LIN {X 0,Y 87.51,Z 409.05,A -85,B 0,C 180,E1 -30606.359,E2 -30606.359} C_VEL
LIN {X 0,Y 79.775,Z 420.472,A -85,B 0,C 180,E1 -30607.649,E2 -30607.649} C_VEL
LIN {X 0,Y 71.234,Z 430.536,A -85,B 0,C 180,E1 -30609.388,E2 -30609.388} C_VEL
LIN {X 0,Y 62.803,Z 438.788,A -85,B 0,C 180,E1 -30611.717,E2 -30611.717} C_VEL
LIN {X 0,Y 52.393,Z 447.262,A -85,B 0,C 180,E1 -30615.825,E2 -30615.825} C_VEL
LIN {X 0,Y 44.908,Z 452.36,A -85,B 0,C 180,E1 -30620.118,E2 -30620.118} C_VEL
LIN {X 0,Y 35.789,Z 457.715,A -85,B 0,C 180,E1 -30627.912,E2 -30627.912} C_VEL
LIN {X 0,Y 27.714,Z 461.88,A -85,B 0,C 180,E1 -30640.469,E2 -30640.469} C_VEL
LIN {X 0,Y 23.498,Z 464.077,A -85,B 0,C 180,E1 -30653.261,E2 -30653.261} C_VEL
LIN {X 0,Y 20.749,Z 465.788,A -85,B 0,C 180,E1 -30670.202,E2 -30670.202} C_VEL
LIN {X 0,Y 20.019,Z 467.089,A -85,B 0,C 180,E1 -30690.001,E2 -30690.001} C_VEL
LIN {X 0,Y 20.814,Z 467.966,A -85,B 0,C 180,E1 -30709.735,E2 -30709.735} C_VEL
LIN {X 0,Y 23.568,Z 468.43,A -85,B 0,C 180,E1 -30726.614,E2 -30726.614} C_VEL
LIN {X 0,Y 33.054,Z 468.146,A -85,B 0,C 180,E1 -30748.265,E2 -30748.265} C_VEL
LIN {X 0,Y 45.111,Z 466.339,A -85,B 0,C 180,E1 -30759.192,E2 -30759.192} C_VEL
LIN {X 0,Y 51.526,Z 464.795,A -85,B 0,C 180,E1 -30762.705,E2 -30762.705} C_VEL
LIN {X 0,Y 63.326,Z 460.995,A -85,B 0,C 180,E1 -30767.176,E2 -30767.176} C_VEL
LIN {X 0,Y 74.89,Z 455.966,A -85,B 0,C 180,E1 -30770.187,E2 -30770.187} C_VEL
LIN {X 0,Y 86.865,Z 449.183,A -85,B 0,C 180,E1 -30772.354,E2 -30772.354} C_VEL
LIN {X 0,Y 97.233,Z 441.823,A -85,B 0,C 180,E1 -30773.643,E2 -30773.643} C_VEL
LIN {X 0,Y 107.631,Z 432.702,A -85,B 0,C 180,E1 -30774.735,E2 -30774.735} C_VEL
LIN {X 0,Y 116.334,Z 423.229,A -85,B 0,C 180,E1 -30775.417,E2 -30775.417} C_VEL
LIN {X 0,Y 124.178,Z 412.736,A -85,B 0,C 180,E1 -30775.957,E2 -30775.957} C_VEL
LIN {X 0,Y 131.301,Z 400.788,A -85,B 0,C 180,E1 -30776.367,E2 -30776.367} C_VEL
LIN {X 0,Y 134.706,Z 393.665,A -85,B 0,C 180,E1 -30776.626,E2 -30776.626} C_VEL
LIN {X 0,Y 135.001,Z 392.963,A -85,B 0,C 180,E1 -30777.016,E2 -30777.016} C_VEL
LIN {X 0,Y 134.921,Z 393.119,A -85,B 0,C 180,E1 -30777.835,E2 -30777.835} C_VEL
LIN {X 0,Y 134.487,Z 394.109,A -85,B 0,C 180,E1 -30778.062,E2 -30778.062} C_VEL
LIN {X 0,Y 128.816,Z 405.217,A -85,B 0,C 180,E1 -30778.474,E2 -30778.474} C_VEL
LIN {X 0,Y 122.13,Z 415.614,A -85,B 0,C 180,E1 -30779.019,E2 -30779.019} C_VEL
LIN {X 0,Y 114.207,Z 425.552,A -85,B 0,C 180,E1 -30779.693,E2 -30779.693} C_VEL
LIN {X 0,Y 105.428,Z 434.57,A -85,B 0,C 180,E1 -30780.7,E2 -30780.7} C_VEL
LIN {X 0,Y 94.932,Z 443.346,A -85,B 0,C 180,E1 -30781.934,E2 -30781.934} C_VEL
LIN {X 0,Y 84.497,Z 450.323,A -85,B 0,C 180,E1 -30783.533,E2 -30783.533} C_VEL
LIN {X 0,Y 74.457,Z 455.749,A -85,B 0,C 180,E1 -30785.637,E2 -30785.637} C_VEL
LIN {X 0,Y 63.956,Z 460.241,A -85,B 0,C 180,E1 -30788.51,E2 -30788.51} C_VEL
LIN {X 0,Y 60.248,Z 461.578,A -85,B 0,C 180,E1 -30789.725,E2 -30789.725} C_VEL
LIN {X 0,Y 54.742,Z 463.267,A -85,B 0,C 180,E1 -30791.162,E2 -30791.162} C_VEL
LIN {X 0,Y 45.104,Z 465.509,A -85,B 0,C 180,E1 -30792.147,E2 -30792.147} C_VEL
LIN {X 0,Y 37.28,Z 466.756,A -85,B 0,C 180,E1 -30793.101,E2 -30793.101} C_VEL
LIN {X 0,Y 31.572,Z 467.361,A -85,B 0,C 180,E1 -30795.483,E2 -30795.483} C_VEL
LIN {X 0,Y 29.771,Z 467.484,A -85,B 0,C 180,E1 -30796.945,E2 -30796.945} C_VEL
LIN {X 0,Y 23.278,Z 467.733,A -85,B 0,C 180,E1 -30805.076,E2 -30805.076} C_VEL
LIN {X 0,Y 17.837,Z 467.52,A -85,B 0,C 180,E1 -30817.998,E2 -30817.998} C_VEL
LIN {X 0,Y 13.915,Z 466.905,A -85,B 0,C 180,E1 -30839.663,E2 -30839.663} C_VEL
LIN {X 0,Y 12.831,Z 465.908,A -85,B 0,C 180,E1 -30869.999,E2 -30869.999} C_VEL
LIN {X 0,Y 15.149,Z 464.523,A -85,B 0,C 180,E1 -30897.64,E2 -30897.64} C_VEL
LIN {X 0,Y 22.348,Z 461.624,A -85,B 0,C 180,E1 -30921.83,E2 -30921.83} C_VEL
LIN {X 0,Y 31.367,Z 457.708,A -85,B 0,C 180,E1 -30933.667,E2 -30933.667} C_VEL
LIN {X 0,Y 41.065,Z 452.666,A -85,B 0,C 180,E1 -30940.268,E2 -30940.268} C_VEL
LIN {X 0,Y 51.081,Z 446.319,A -85,B 0,C 180,E1 -30944.385,E2 -30944.385} C_VEL
LIN {X 0,Y 61.273,Z 438.386,A -85,B 0,C 180,E1 -30947.147,E2 -30947.147} C_VEL
LIN {X 0,Y 69.817,Z 430.311,A -85,B 0,C 180,E1 -30948.949,E2 -30948.949} C_VEL
LIN {X 0,Y 78.417,Z 420.461,A -85,B 0,C 180,E1 -30950.35,E2 -30950.35} C_VEL
LIN {X 0,Y 86.175,Z 409.383,A -85,B 0,C 180,E1 -30951.437,E2 -30951.437} C_VEL
LIN {X 0,Y 92.915,Z 397.136,A -85,B 0,C 180,E1 -30952.225,E2 -30952.225} C_VEL
LIN {X 0,Y 97.715,Z 385.779,A -85,B 0,C 180,E1 -30952.782,E2 -30952.782} C_VEL
LIN {X 0,Y 101.726,Z 372.53,A -85,B 0,C 180,E1 -30953.267,E2 -30953.267} C_VEL
LIN {X 0,Y 103.028,Z 366.567,A -85,B 0,C 180,E1 -30953.488,E2 -30953.488} C_VEL
LIN {X 0,Y 103.038,Z 365.719,A -85,B 0,C 180,E1 -30956.089,E2 -30956.089} C_VEL
LIN {X 0,Y 103.054,Z 365.939,A -85,B 0,C 180,E1 -30958.778,E2 -30958.778} C_VEL
LIN {X 0,Y 103.087,Z 366.426,A -85,B 0,C 180,E1 -30960.243,E2 -30960.243} C_VEL
LIN {X 0,Y 99.984,Z 379.167,A -85,B 0,C 180,E1 -30960.627,E2 -30960.627} C_VEL
LIN {X 0,Y 96.34,Z 389.562,A -85,B 0,C 180,E1 -30960.864,E2 -30960.864} C_VEL
LIN {X 0,Y 91.387,Z 400.467,A -85,B 0,C 180,E1 -30961.301,E2 -30961.301} C_VEL
LIN {X 0,Y 84.384,Z 412.413,A -85,B 0,C 180,E1 -30961.942,E2 -30961.942} C_VEL
LIN {X 0,Y 76.523,Z 423.065,A -85,B 0,C 180,E1 -30962.834,E2 -30962.834} C_VEL
LIN {X 0,Y 68.683,Z 431.762,A -85,B 0,C 180,E1 -30963.911,E2 -30963.911} C_VEL
LIN {X 0,Y 60.024,Z 439.78,A -85,B 0,C 180,E1 -30965.596,E2 -30965.596} C_VEL
LIN {X 0,Y 49.735,Z 447.623,A -85,B 0,C 180,E1 -30968.444,E2 -30968.444} C_VEL
LIN {X 0,Y 42.983,Z 451.954,A -85,B 0,C 180,E1 -30971.179,E2 -30971.179} C_VEL
LIN {X 0,Y 33.06,Z 457.351,A -85,B 0,C 180,E1 -30976.941,E2 -30976.941} C_VEL
LIN {X 0,Y 23.703,Z 461.553,A -85,B 0,C 180,E1 -30987.188,E2 -30987.188} C_VEL
LIN {X 0,Y 18.295,Z 463.782,A -85,B 0,C 180,E1 -30999.798,E2 -30999.798} C_VEL
LIN {X 0,Y 14.252,Z 465.516,A -85,B 0,C 180,E1 -31020.454,E2 -31020.454} C_VEL
LIN {X 0,Y 12.925,Z 466.835,A -85,B 0,C 180,E1 -31050.001,E2 -31050.001} C_VEL
LIN {X 0,Y 14.326,Z 467.728,A -85,B 0,C 180,E1 -31079.38,E2 -31079.38} C_VEL
LIN {X 0,Y 18.349,Z 468.221,A -85,B 0,C 180,E1 -31100,E2 -31100} C_VEL
LIN {X 0,Y 29.924,Z 467.974,A -85,B 0,C 180,E1 -31119.958,E2 -31119.958} C_VEL
LIN {X 0,Y 43.095,Z 466.208,A -85,B 0,C 180,E1 -31128.095,E2 -31128.095} C_VEL
LIN {X 0,Y 49.876,Z 464.69,A -85,B 0,C 180,E1 -31130.529,E2 -31130.529} C_VEL
LIN {X 0,Y 61.317,Z 461.223,A -85,B 0,C 180,E1 -31133.419,E2 -31133.419} C_VEL
LIN {X 0,Y 73.483,Z 456.181,A -85,B 0,C 180,E1 -31135.555,E2 -31135.555} C_VEL
LIN {X 0,Y 84.463,Z 450.3,A -85,B 0,C 180,E1 -31136.862,E2 -31136.862} C_VEL
LIN {X 0,Y 91.454,Z 445.758,A -85,B 0,C 180,E1 -31137.455,E2 -31137.455} C_VEL
LIN {X 0,Y 91.424,Z 445.765,A -85,B 0,C 180,E1 -31137.935,E2 -31137.935} C_VEL
LIN {X 0,Y 80.833,Z 452.325,A -85,B 0,C 180,E1 -31139.076,E2 -31139.076} C_VEL
LIN {X 0,Y 70.285,Z 457.525,A -85,B 0,C 180,E1 -31140.698,E2 -31140.698} C_VEL
LIN {X 0,Y 58.328,Z 462.003,A -85,B 0,C 180,E1 -31143.151,E2 -31143.151} C_VEL
LIN {X 0,Y 49.444,Z 464.5,A -85,B 0,C 180,E1 -31145.735,E2 -31145.735} C_VEL
LIN {X 0,Y 38.674,Z 466.568,A -85,B 0,C 180,E1 -31150.471,E2 -31150.471} C_VEL
LIN {X 0,Y 29.771,Z 467.484,A -85,B 0,C 180,E1 -31156.945,E2 -31156.945} C_VEL
LIN {X 0,Y 24.313,Z 467.809,A -85,B 0,C 180,E1 -31161.701,E2 -31161.701} C_VEL
LIN {X 0,Y 14.878,Z 467.626,A -85,B 0,C 180,E1 -31170.865,E2 -31170.865} C_VEL
LIN {X 0,Y 7.959,Z 466.869,A -85,B 0,C 180,E1 -31191.717,E2 -31191.717} C_VEL
LIN {X 0,Y 5.928,Z 466.01,A -85,B 0,C 180,E1 -31239.221,E2 -31239.221} C_VEL
LIN {X 0,Y 6.619,Z 465.601,A -85,B 0,C 180,E1 -31255.999,E2 -31255.999} C_VEL
LIN {X 0,Y 15.545,Z 462.994,A -85,B 0,C 180,E1 -31294.712,E2 -31294.712} C_VEL
LIN {X 0,Y 25.53,Z 459.472,A -85,B 0,C 180,E1 -31304.469,E2 -31304.469} C_VEL
LIN {X 0,Y 35.798,Z 454.855,A -85,B 0,C 180,E1 -31308.996,E2 -31308.996} C_VEL
LIN {X 0,Y 47.908,Z 447.891,A -85,B 0,C 180,E1 -31311.973,E2 -31311.973} C_VEL
LIN {X 0,Y 58.354,Z 440.351,A -85,B 0,C 180,E1 -31313.514,E2 -31313.514} C_VEL
LIN {X 0,Y 67.067,Z 432.647,A -85,B 0,C 180,E1 -31314.567,E2 -31314.567} C_VEL
LIN {X 0,Y 76.671,Z 422.176,A -85,B 0,C 180,E1 -31315.452,E2 -31315.452} C_VEL
LIN {X 0,Y 84.535,Z 411.521,A -85,B 0,C 180,E1 -31316.069,E2 -31316.069} C_VEL
LIN {X 0,Y 90.656,Z 401.199,A -85,B 0,C 180,E1 -31316.485,E2 -31316.485} C_VEL
LIN {X 0,Y 91.53,Z 399.474,A -85,B 0,C 180,E1 -31316.542,E2 -31316.542} C_VEL
LIN {X 0,Y 91.503,Z 399.537,A -85,B 0,C 180,E1 -31316.84,E2 -31316.84} C_VEL
LIN {X 0,Y 85.325,Z 410.339,A -85,B 0,C 180,E1 -31317.074,E2 -31317.074} C_VEL
LIN {X 0,Y 77.386,Z 421.345,A -85,B 0,C 180,E1 -31317.431,E2 -31317.431} C_VEL
LIN {X 0,Y 68.567,Z 431.194,A -85,B 0,C 180,E1 -31317.952,E2 -31317.952} C_VEL
LIN {X 0,Y 59.752,Z 439.272,A -85,B 0,C 180,E1 -31318.751,E2 -31318.751} C_VEL
LIN {X 0,Y 49.196,Z 447.192,A -85,B 0,C 180,E1 -31320.183,E2 -31320.183} C_VEL
LIN {X 0,Y 42.186,Z 451.549,A -85,B 0,C 180,E1 -31321.665,E2 -31321.665} C_VEL
LIN {X 0,Y 31.723,Z 456.985,A -85,B 0,C 180,E1 -31324.495,E2 -31324.495} C_VEL
LIN {X 0,Y 21.402,Z 461.225,A -85,B 0,C 180,E1 -31329.896,E2 -31329.896} C_VEL
LIN {X 0,Y 14.781,Z 463.48,A -85,B 0,C 180,E1 -31338.027,E2 -31338.027} C_VEL
LIN {X 0,Y 8.794,Z 465.244,A -85,B 0,C 180,E1 -31356.949,E2 -31356.949} C_VEL
LIN {X 0,Y 5.819,Z 466.58,A -85,B 0,C 180,E1 -31410.003,E2 -31410.003} C_VEL
LIN {X 0,Y 8.839,Z 467.489,A -85,B 0,C 180,E1 -31462.668,E2 -31462.668} C_VEL
LIN {X 0,Y 14.815,Z 468.007,A -85,B 0,C 180,E1 -31481.583,E2 -31481.583} C_VEL
LIN {X 0,Y 28.286,Z 467.801,A -85,B 0,C 180,E1 -31493.649,E2 -31493.649} C_VEL
LIN {X 0,Y 42.205,Z 466.072,A -85,B 0,C 180,E1 -31497.613,E2 -31497.613} C_VEL
LIN {X 0,Y 42.178,Z 466.055,A -85,B 0,C 180,E1 -31498.743,E2 -31498.743} C_VEL
LIN {X 0,Y 35.142,Z 467.067,A -85,B 0,C 180,E1 -31500.561,E2 -31500.561} C_VEL
LIN {X 0,Y 21.257,Z 467.924,A -85,B 0,C 180,E1 -31507.308,E2 -31507.308} C_VEL
LIN {X 0,Y 14.56,Z 467.745,A -85,B 0,C 180,E1 -31515.112,E2 -31515.112} C_VEL
LIN {X 0,Y 8.534,Z 467.147,A -85,B 0,C 180,E1 -31534.555,E2 -31534.555} C_VEL
LIN {X 0,Y 6.619,Z 465.601,A -85,B 0,C 180,E1 -31615.999,E2 -31615.999} C_VEL
LIN {X 0,Y 8.105,Z 467.565,A -85,B 0,C 180,E1 -31630.582,E2 -31630.582} C_VEL
LIN {X 0,Y 8.105,Z 600,A -85,B 0,C 180,E1 -31630.582,E2 -31630.582} C_VEL
LIN {X 0,Y 8.105,Z 600,A -85,B 0,C 180,E1 -31630.582,E2 -31630.582}

QRS_NEXT_CUT()

QRS_NEXT()
QRS_HOME()

END
